PROGRAM FAST
VAR
		VeloConvert  	:LREAL;
		EncoderUdint	:UDINT;
		test			:BOOL;
		
		
END_VAR



VeloConvert := ((RealVelocimeterD / 250.0000000)/10);



EncoderD := (yAxis.NcToPlc.ActPos *( -1.00)) /10 ;



test;

END_PROGRAM

(* stored: Version 1.1.0.1, ProductVersion 3.1.4024.12
   POU FAST: Id {a373178b-a3f5-45aa-8fdd-f702d1165cf0}, SpecialFunc None *)
